// TIA Portal V20 export
TYPE "typeAxisActuatorCondition"
// stored: Access Published, Namespace LER
   STRUCT
      Home_INT : Bool;
      Work_INT : Bool;
      Home_INT_Error : Bool;
      Work_INT_Error : Bool;
      intOut : Array[0..9] of Bool;
   END_STRUCT;
END_TYPE
